TYPE BallSeat_IO_typ:
STRUCT
	Inputs	: Orient_Inputs_typ;
	Outputs	: Orient_Outputs_typ;
END_STRUCT
END_TYPE

(* stored: Version 1.1.0.1, ProductVersion 3.1.4024.12
   DUT BallSeat_IO_typ: Id {c93c3448-3f85-03a0-1da5-2260c635e3e1} *)
